Xinje XCPPro project, PLC1: XC3-32 (software 3.3k)

PROGRAM Ladder

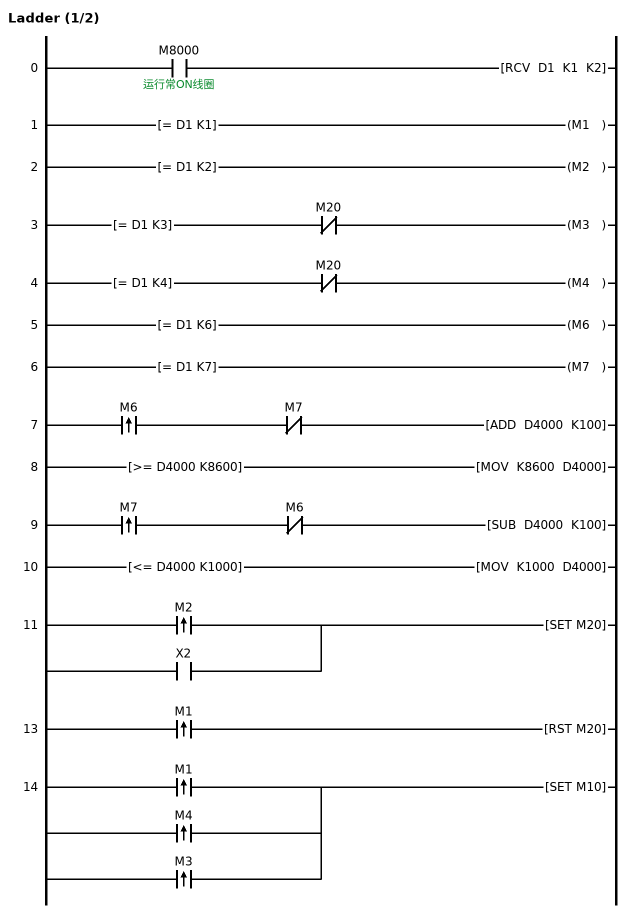
LD     M8000	; 运行常ON线圈
RCV    D1 K1 K2
LD=    D1 K1
OUT    M1
LD=    D1 K2
OUT    M2
LD=    D1 K3
ANI    M20
OUT    M3
LD=    D1 K4
ANI    M20
OUT    M4
LD=    D1 K6
OUT    M6
LD=    D1 K7
OUT    M7
LDP    M6
ANI    M7
ADD    D4000 K100
LD>=   D4000 K8600
MOV    K8600 D4000
LDP    M7
ANI    M6
SUB    D4000 K100
LD<=   D4000 K1000
MOV    K1000 D4000
LDP    M2
OR     X2
SET    M20
LDP    M1
RST    M20
LDP    M1
ORP    M4
ORP    M3
SET    M10

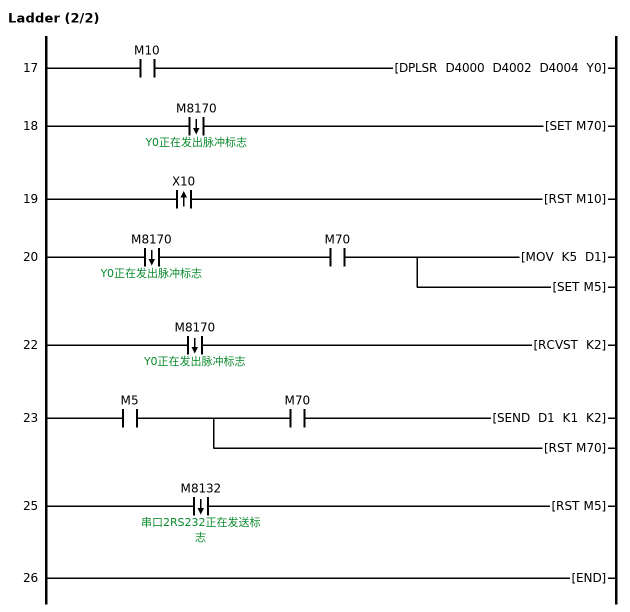
LD     M10
DPLSR  D4000 D4002 D4004 Y0
LDF    M8170	; Y0正在发出脉冲标志
SET    M70
LDP    X10
RST    M10
LDF    M8170	; Y0正在发出脉冲标志
AND    M70
MOV    K5 D1
SET    M5
LDF    M8170	; Y0正在发出脉冲标志
RCVST  K2
LD     M5
MPS
AND    M70
SEND   D1 K1 K2
MPP
RST    M70
LDF    M8132	; 串口2RS232正在发送标志
RST    M5
END